{attribute 'linkalways'} 
{attribute 'no_explicit_call' := 'This FB is a CLASS and must be accessed using methods or properties'}
{attribute 'enable_dynamic_creation'}
FUNCTION_BLOCK Node_F_VN_FillContainer_TcVnVector3_UINT EXTENDS VisionNode
VAR
    ipContainer : _ITcVnContainer;
    aValue : _TcVnVector3_UINT;
    hrPrev : _HRESULT(S_OK);
    hresult : _HRESULT(S_OK);
END_VAR

METHOD PUBLIC  Clone : I_Node
VAR
    pNode : POINTER TO Node_F_VN_FillContainer_TcVnVector3_UINT;
END_VAR
pNode := __NEW(Node_F_VN_FillContainer_TcVnVector3_UINT);
Clone := pNode^;
END_METHOD

METHOD FB_init : BOOL
VAR_INPUT
    bInitRetains : BOOL; // if TRUE, the retain variables are initialized (warm start / cold start)
    bInCopyCode : BOOL;  // if TRUE, the instance afterwards gets moved into the copy code (online change)
END_VAR
AddInput('ipContainer', ipContainer);
AddInput('aValue', aValue);
AddInput('hrPrev', hrPrev);
AddOutput('ipContainer', ipContainer);
AddOutput('hresult',hresult);
END_METHOD

METHOD PROTECTED OnExecute
hresult.Value := F_VN_FillContainer_TcVnVector3_UINT(
    ipContainer := ipContainer.Value,
    aValue := aValue.Value,
    hrPrev:= hrPrev.Value);
END_METHOD

METHOD PUBLIC PreExecutionCheck
VAR_INPUT
    Check : I_PreExecutionChecks;
END_VAR
Check.IsTrue(ipContainer.IsValid, 'ipContainer must be a valid container');
Check.IsTrue(ipContainer.IsType(TC_GLOBAL_CONST_LIST.ContainerType_Vector_TcVnVector3_UINT), 'ipContainer contains incorrect type');
END_METHOD

END_FUNCTION_BLOCK

(* stored: Version 1.1.0.1, ProductVersion 3.1.4026.13
   POU Node_F_VN_FillContainer_TcVnVector3_UINT: Id {e98fe359-96b9-4e58-a61d-ee9501cdfce5}, SpecialFunc None
   Folder Constructor: Id {ff2e3ef6-d7c1-44bc-9a28-e2f35a8e18ba}
   Method Clone: Id {4ba76e4a-9b9b-4f95-bdc8-3a3001f8652c}
   Method FB_init: Id {74b5e363-f7ef-483b-93ad-41ed92fd20c1}
   Method OnExecute: Id {00a51ba6-3852-47bf-9c9f-257e67df6bc6}
   Method PreExecutionCheck: Id {7f34c2be-61cf-41ff-84fb-919a9b392461} *)
